SUBAPPLICATION Uebung_010d_PC_A_OPC (* Geraet A (Station 11, 192.168.1.11): SoftKey_F1-Tastendruck (SK_RELEASED) ruft per CLIENT_0 einen argument- und rueckgabewertlosen OPC-UA-Methodenaufruf auf Geraet B auf (reiner RPC-Trigger, kein Wertwechsel-Trick noetig, kein AX_T_FF auf diesem Geraet); GreenWhiteBackground zeigt den von Geraet B lokal ueberwachten Flipflop-Zustand - 'SUB style': das Protokoll steckt im MyLib::sys-Composite, nicht in der Resource des Geraets *)
  (* Standard: 61499-2; Description: Copyright (c) 2026 Meisterschulen am Ostbahnhof This program and the accompanying materials are made available under the terms of the Eclipse Public License 2.0 which is available at https://www.eclipse.org/legal/epl-2.0/ SPDX-License-Identifier: EPL-2.0 *)
  (* Version 1.0, 2026-09-02, Franz Höpfinger, Meisterschulen am Ostbahnhof, initial API and implementation and/or initial documentation *)
  PACKAGE MyLib::sys;
  IMPORT isobus::UT::Q::const::IDs::ID_NULL;
  IMPORT isobus::UT::io::Softkey::SoftKeyActivationCode::SK_RELEASED;
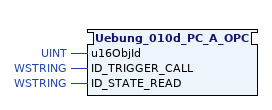
  VAR_INPUT
    u16ObjId : UINT := ID_NULL; (* Object ID Softkey/Background *)
    ID_TRIGGER_CALL : WSTRING; (* Remote-Methodenadresse (ACTION=CALL_METHOD) fuer den argumentlosen Trigger-Methodenaufruf auf Geraet B *)
    ID_STATE_READ : WSTRING; (* Lokal ueberwachte Adresse (BOOL, ACTION=READ) fuer den Flipflop-Zustand, wird von Geraet B remote beschrieben *)
  END_VAR
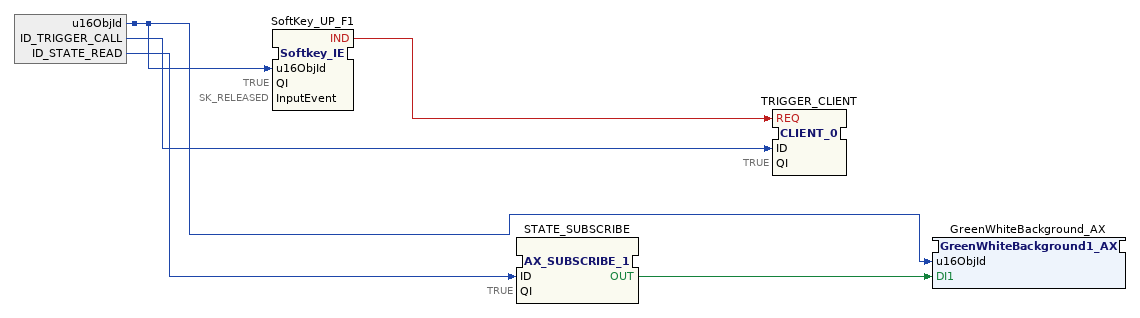
  FBS
    SoftKey_UP_F1 : isobus::UT::io::Softkey::Softkey_IE(QI := TRUE, InputEvent := SK_RELEASED);
    TRIGGER_CLIENT : iec61499::net::CLIENT_0(QI := TRUE);
    STATE_SUBSCRIBE : adapter::net::AX_SUBSCRIBE_1(QI := TRUE);
  END_FBS
  SUBAPPS
    GreenWhiteBackground_AX : MyLib::sys::GreenWhiteBackground1_AX;
  END_SUBAPPS
  EVENT_CONNECTIONS
    SoftKey_UP_F1.IND TO TRIGGER_CLIENT.REQ;
  END_CONNECTIONS
  DATA_CONNECTIONS
    u16ObjId TO SoftKey_UP_F1.u16ObjId;
    u16ObjId TO GreenWhiteBackground_AX.u16ObjId;
    ID_TRIGGER_CALL TO TRIGGER_CLIENT.ID;
    ID_STATE_READ TO STATE_SUBSCRIBE.ID;
  END_CONNECTIONS
  ADAPTER_CONNECTIONS
    STATE_SUBSCRIBE.OUT TO GreenWhiteBackground_AX.DI1;
  END_CONNECTIONS
END_SUBAPPLICATION
